// TIA Portal V19 export
FUNCTION_BLOCK "NetworkSwitchFaceplate"   // FB11, LAD
{ S7_Optimized_Access := 'TRUE' }
// stored: MemoryReserve 100, SetENOAutomatically false
   VAR_INPUT
      Index : Int;
   END_VAR
   VAR_OUTPUT
      PeerName { ExternalAccessible := 'False'; ExternalVisible := 'False'; ExternalWritable := 'False'} : String;
   END_VAR
   VAR_IN_OUT
      Port : "NetworkSwitchHMI";
   END_VAR
BEGIN

REGION Network 1 (SCL): Move all IN/OUT variables into Static values based on index selected from HMI

   #Port.Port := #Port.Ports[#Index];
END_REGION
END_FUNCTION_BLOCK
